/// MODE to run (inside of MODULE_INTERFACE_INPUT)
TYPE DUT_MODE :
(
	///Initialitzation number mode
	Init := 0,
	///Automatic number mode
	Auto := 1,
	///Manual number mode
	Manual := 2,
	Reset := 3
);
END_TYPE

(* stored: Version 1.1.0.1, ProductVersion 3.1.0.25
   DUT DUT_MODE: Id {68ff4b77-c15d-40ad-8643-4ecec7363ccb} *)
